// TIA Portal V18 export
// export: Created 2025-12-01T17:53:03.7409904Z, ExportSetting None, DisplayName Totally Integrated Automation Portal, DisplayVersion V18 Update 5, DisplayName TIA Portal Openness, DisplayVersion V18 Update 5, DisplayName TIA Portal Teamcenter Gateway, DisplayVersion V18, DisplayName TIA Portal Version Control Interface, DisplayVersion V18, DisplayName STEP 7 Professional, DisplayVersion V18 Update 5, DisplayName STEP 7 Safety, DisplayVersion V18, DisplayName WinCC Professional, DisplayVersion V18 Update 5
Screen "266_Cylinder_H3"  1280x800, Number=266, Template=02ManualUnit1
  ScreenLayer "Layer_0"
    FaceplateInstance "Cylinder_S71500_TP700_1" at 0,85 size 1279x80  FaceplateTypeName=03 FunctionBlocks@$@101 Cylinder@$@101.2 HMI@$@S7-1500@$@Cylinder_S71500_TP700 V 0.0.29
      Cy := STxxxCylinder027
      CylinderName := Cyl name
      HomeButtonName := Cyl go home button
      WorkButtonName := Cyl go work button
      HomeQaddress := Cyl home Q
      HomeIaddress := Cyl home I
      WorkIaddress := Cyl work I
      WorkQaddress := Cyl work Q
    FaceplateInstance "Cylinder_S71500_TP700_3" at 0,160 size 1279x80  FaceplateTypeName=03 FunctionBlocks@$@101 Cylinder@$@101.2 HMI@$@S7-1500@$@Cylinder_S71500_TP700 V 0.0.29
      Cy := STxxxCylinder028
      CylinderName := Cyl name
      HomeButtonName := Cyl go home button
      WorkButtonName := Cyl go work button
      HomeQaddress := Cyl home Q
      HomeIaddress := Cyl home I
      WorkIaddress := Cyl work I
      WorkQaddress := Cyl work Q
    FaceplateInstance "Cylinder_S71500_TP700_2" at 0,235 size 1279x80  FaceplateTypeName=03 FunctionBlocks@$@101 Cylinder@$@101.2 HMI@$@S7-1500@$@Cylinder_S71500_TP700 V 0.0.29
      Cy := STxxxCylinder029
      CylinderName := Cyl name
      HomeButtonName := Cyl go home button
      WorkButtonName := Cyl go work button
      HomeQaddress := Cyl home Q
      HomeIaddress := Cyl home I
      WorkIaddress := Cyl work I
      WorkQaddress := Cyl work Q
    Button "btnMenu6" at 640,725 size 128x75  TextOff="H-气缸3 / H-Cylinder3", TextOn="H-气缸3 / H-Cylinder3"
      on Click: ActivateScreen(Screen name := , Object number := 0)
    Button "按钮_9" at 128,725 size 128x75  PictureOff=向右箭头_0, TextOff="H-气缸1 / H-Cylinder1", TextOn="H-气缸1 / H-Cylinder1"
      on Click: ActivateScreen(Screen name := 260_Cylinder_H1, Object number := 0)
    Button "btnMenu4" at 384,725 size 128x75  TextOff="H-气缸2 / H-Cylinder2", TextOn="H-气缸2 / H-Cylinder2"
      on Click: ActivateScreen(Screen name := 263_Cylinder_H2, Object number := 0)
    Button "btnMenu5" at 512,725 size 128x75  TextOff="H-电机2 / H-Motor2", TextOn="H-电机2 / H-Motor2"
      on Click: ActivateScreen(Screen name := 264_Motor_H2, Object number := 0)
    Button "btnMenu7" at 896,725 size 128x75
    Button "btnMenu6_2" at 768,725 size 128x75  TextOff="H-电机3 / H-Motor3", TextOn="H-电机3 / H-Motor3"
      on Click: ActivateScreen(Screen name := 267_Motor_H3, Object number := 0)
    Button "btnMenu7_1" at 1024,725 size 128x75
    Button "btnMenu4_1" at 256,725 size 128x75  TextOff="H-电机1 / H-Motor1", TextOn="H-电机1 / H-Motor1"
      on Click: ActivateScreen(Screen name := 261_Motor_H1, Object number := 0)
